(* IEC 61131-3 sources: AXOpen/src/components.festo.drives/ctrl/src/AxoCmmtAs (part 4) *)

            _AxisReference ?= AxisRef;

            IF(_AxisReference = NULL) THEN
                Messenger.Activate(     UINT#1690, eAxoMessageCategory#ProgrammingError);
                DriveStatus.Error.Id := UINT#1690;
                RETURN;
            END_IF;

            IF Enable THEN
                THIS.UpdateInputs(AxisRef);
                Valid := TRUE;
                Torque := THIS.ActualTorque;
            END_IF;
        END_METHOD

        ///<summary>
        /// This method returns in detail the status of the state diagram of the axis
        ///</summary>
        VAR INTERNAL
            MC_ReadStatusEnable_PV				: 	BOOL := FALSE;		//Enable - previous value
            MC_ReadStatusDone_PV				:	BOOL := FALSE;		//Done - previous value
            MC_ReadStatusStateNumber			: 	INT; 				//Call number of the method MC_ReadRealParameter
        END_VAR
        METHOD PUBLIC OVERRIDE MC_ReadStatus
            VAR_INPUT
                AxisRef             :   AXOpen.Components.Abstractions.Drives.IAxoAxisReference;
                Enable              :   BOOL;                       //  Get the value of the parameter continuously while enabled
            END_VAR
            VAR_OUTPUT
                Valid               :   BOOL;                       //  A valid output is available at the method
                Busy                :   BOOL;                       //  The method is not finished and new output values are to be expected
                Error               :   BOOL;                       //  Signals that an error has occurred within the method
                ErrorID             :   DINT;                       //  Error identification
                ErrorStop           :   BOOL;                       //  See state diagram
                Disabled            :   BOOL;                       //  See state diagram
                Stopping            :   BOOL;                       //  See state diagram
                Homing              :   BOOL;                       //  See state diagram
                Standstill          :   BOOL;                       //  See state diagram
                DiscreteMotion      :   BOOL;                       //  See state diagram
                ContinuousMotion    :   BOOL;                       //  See state diagram
                SynchronizedMotion  : BOOL;                       //  See state diagram
            END_VAR
            VAR
                _AxisReference :  REF_TO AXOpen.Components.Festo.Drives.AxoCmmtAsAxisReference;
                Dummy : BOOL;
            END_VAR

            _AxisReference ?= AxisRef;

            IF(_AxisReference = NULL) THEN
                Messenger.Activate(     UINT#1700, eAxoMessageCategory#ProgrammingError);
                DriveStatus.Error.Id := UINT#1700;
                RETURN;
            END_IF;

            IF Enable THEN
                THIS.UpdateInputs(AxisRef);
                Valid := TRUE;
                Error                   := _AxisReference^.Telegram111_In.ZSW1.faultPresent;
                ErrorID                 := _AxisReference^.Telegram111_In.Fault_Code;
                ErrorStop               := DriveState = AXOpen.Components.Drives.eAxoDriveState#ErrorStop;;
                Disabled                := DriveState = AXOpen.Components.Drives.eAxoDriveState#Disabled;
                Stopping                := DriveState = AXOpen.Components.Drives.eAxoDriveState#Stopping;
                Homing                  := DriveState = AXOpen.Components.Drives.eAxoDriveState#Homing;
                Standstill              := DriveState = AXOpen.Components.Drives.eAxoDriveState#Standstill;
                DiscreteMotion          := DriveState = AXOpen.Components.Drives.eAxoDriveState#DiscreteMotion;
                ContinuousMotion        := DriveState = AXOpen.Components.Drives.eAxoDriveState#ContinuousMotion;
                SynchronizedMotion      := DriveState = AXOpen.Components.Drives.eAxoDriveState#SynchronizedMotion;
            END_IF;
        END_METHOD

        ///<summary>
        /// This method returns in detail the status of the axis with respect to the motion currently in progress.
        ///</summary>
        VAR INTERNAL
            MC_ReadMotionStateEnable_PV     : 	BOOL := FALSE;		//Enable - previous value
            MC_ReadMotionStateErrorID       : 	WORD;
            MC_ReadMotionStateCycle			: 	ULINT;
            MC_ReadMotionStateValue			: 	LINT;
            MC_ReadMotionStateValid			: 	BOOL;
        END_VAR
        METHOD PUBLIC OVERRIDE MC_ReadMotionState
            VAR_INPUT
                AxisRef         :   AXOpen.Components.Abstractions.Drives.IAxoAxisReference;
                Enable          :   BOOL;                       //  Get the value of the parameter continuously while enabled
                Source          :   AXOpen.Components.Abstractions.Drives.eAxoSource;                 //  Defines the source of the relevant data: CommandedValue;SetValue, ActualValue.
            END_VAR
            VAR_OUTPUT
                Valid           :   BOOL;                       //  A valid output is available at the method
                Busy            :   BOOL;                       //  The method is not finished and new output values are to be expected
                Error           :   BOOL;                       //  Signals that an error has occurred within the method
                ErrorID         :   DINT;                       //  Error identification
                ConstantVelocity:   BOOL;                       //  Velocity is constant. Velocity may be 0. For the actual value a window is applicable (window is vendor specific)
                Accelerating    :   BOOL;                       //  Increasing the absolute value of the velocity
                Decelerating    :   BOOL;                       //  Decreasing the absolute value of the velocity
                DirectionPositive:  BOOL;                       //  Signals that the position is increasing
                DirectionNegative:  BOOL;                       //  Signals that the position is decreasing
            END_VAR
            VAR
                _AxisReference :  REF_TO AXOpen.Components.Festo.Drives.AxoCmmtAsAxisReference;
                Dummy : BOOL;
            END_VAR

            _AxisReference ?= AxisRef;

            IF(_AxisReference = NULL) THEN
                Messenger.Activate(     UINT#1710, eAxoMessageCategory#ProgrammingError);
                DriveStatus.Error.Id := UINT#1710;
                RETURN;
            END_IF;

            IF Enable THEN
                THIS.UpdateInputs(AxisRef);
                Valid := TRUE;
                Error                   := _AxisReference^.Telegram111_In.ZSW1.faultPresent;
                ErrorID                 := _AxisReference^.Telegram111_In.Fault_Code;
                ConstantVelocity        := FALSE;
                Accelerating            := _AxisReference^.Telegram111_In.ZSW1.axisAccelerates;
                Decelerating            := _AxisReference^.Telegram111_In.ZSW1.axisDecelerates;
                DirectionPositive       := _AxisReference^.Telegram111_In.POS_ZSW2.%X4;
                DirectionNegative       := _AxisReference^.Telegram111_In.POS_ZSW2.%X5;
             END_IF;
        END_METHOD

        ///<summary>
        /// This method reads information concerning an axis, like modes, inputs directly related to the axis,
        /// and certain status information.
        ///<summary>
        METHOD PUBLIC OVERRIDE MC_ReadAxisInfo
            VAR_INPUT
                AxisRef             :   AXOpen.Components.Abstractions.Drives.IAxoAxisReference;
                Enable              :   BOOL;                       //  Get the value of the parameter continuously while enabled
            END_VAR
            VAR_OUTPUT
                Valid               :   BOOL;                       //  A valid output is available at the method
                Busy                :   BOOL;                       //  The method is not finished and new output values are to be expected
                Error               :   BOOL;                       //  Signals that an error has occurred within the method
                ErrorID             :   DINT;                       //  Error identification
                HomeAbsSwitch       :   BOOL;                       //  Digital home switch input is active
                LimitSwitchPos      :   BOOL;                       //  Positive hardware end switch is active
                LimitSwitchNeg      :   BOOL;                       //  Negative hardware end switch is active
                Simulation          :   BOOL;                       //  Axis is in simulation mode (e.g. motor is simulated)
                CommunicationReady  :   BOOL;                         //  “Network” is initialized and ready for communication
                ReadyForPowerOn     :   BOOL;                       //  Drive is ready to be enabled (power on)
                PowerOn             :   BOOL;                       //  If TRUE shows that the power stage is switched ON
                IsHomed             :   BOOL;                       //  The absolute reference position is known for the axis (axis is homed)
                AxisWarning         :   BOOL;                       //  Warning(s) on the axis is present
            END_VAR
            VAR
                _AxisReference :  REF_TO AXOpen.Components.Festo.Drives.AxoCmmtAsAxisReference;
                Dummy : BOOL;
            END_VAR

            _AxisReference ?= AxisRef;

            IF(_AxisReference = NULL) THEN
                Messenger.Activate(     UINT#1720, eAxoMessageCategory#ProgrammingError);
                DriveStatus.Error.Id := UINT#1720;
                RETURN;
            END_IF;

            IF Enable THEN
                THIS.UpdateInputs(AxisRef);
                Valid := TRUE;
                Error                   := _AxisReference^.Telegram111_In.ZSW1.faultPresent;
                ErrorID                 := _AxisReference^.Telegram111_In.Fault_Code;
                HomeAbsSwitch           := FALSE;
                LimitSwitchPos          := _AxisReference^.Telegram111_In.POS_ZSW1.%X9;
                LimitSwitchNeg          := _AxisReference^.Telegram111_In.POS_ZSW1.%X8;
                Simulation              := FALSE;
                CommunicationReady      := FALSE;
                ReadyForPowerOn         := _AxisReference^.Telegram111_In.ZSW1.readyForSwitchOn;
                PowerOn                 := _AxisReference^.Telegram111_In.ZSW1.operationEnabled;
                IsHomed                 := _AxisReference^.Telegram111_In.ZSW1.homePosSet;
                AxisWarning             := _AxisReference^.Telegram111_In.ZSW1.warningActive;
            END_IF;
        END_METHOD

        ///<summary>
        /// This method presents general axis errors not relating to the methods.
        /// (for instance axis errors, drive errors, communication errors)
        ///</summary>
        VAR INTERNAL
            MC_ReadAxisErrorEnable_PV        : 	BOOL := FALSE;		//Enable - previous value
            MC_ReadAxisErrorErrorID          : 	DINT;
            MC_ReadAxisErrorCycle			: 	ULINT;
            MC_ReadAxisErrorValue			: 	LINT;
            MC_ReadAxisErrorValid			: 	BOOL;
            LastMessageCode :   ULINT;
        END_VAR
        METHOD PUBLIC OVERRIDE MC_ReadAxisError
            VAR_INPUT
                AxisRef         :   AXOpen.Components.Abstractions.Drives.IAxoAxisReference;
                Enable          :   BOOL;                       //  Get the value of the parameter continuously while enabled
            END_VAR
            VAR_OUTPUT
                Valid           :   BOOL;                       //  A valid output is available at the method
                Busy            :   BOOL;                       //  The method is not finished and new output values are to be expected
                Error           :   BOOL;                       //  Signals that an error has occurred within the method
                ErrorID         :   DINT;                       //  Error identification
                AxisErrorID     :   DWORD;                      //  The value of the axis error. These values are vendor specific
            END_VAR
            VAR
                _AxisReference :  REF_TO AXOpen.Components.Festo.Drives.AxoCmmtAsAxisReference;
                Dummy : BOOL;
                _category  :   AXOpen.Messaging.eAxoMessageCategory;
            END_VAR

            _AxisReference ?= AxisRef;

            IF(_AxisReference = NULL) THEN
                Messenger.Activate(     UINT#1730, eAxoMessageCategory#ProgrammingError);
                DriveStatus.Error.Id := UINT#1730;
                RETURN;
            END_IF;

            IF Enable AND NOT MC_ReadAxisErrorEnable_PV AND State = UINT#0 THEN
                _AxisReference^.Status.CurrentMotionTaskId := AXOpen.Components.Drives.eAxoMotionTaskId#Axo_ReadAxisError;
                _AxisReference^.Data.Cycle := _AxisReference^.Data.Cycle + ULINT#2;
                MC_ReadAxisErrorCycle := _AxisReference^.Data.Cycle ;
            END_IF;

            IF Enable THEN
                THIS.UpdateInputs(AxisRef);
                IF State = UINT#0 THEN
                    Busy := TRUE;
                    MC_ReadAxisErrorErrorID := DINT#0;
                    Parametrization.Inputs.Enable := FALSE;
                    State := UINT#310;
                END_IF;
                IF State = UINT#310 THEN
                    Busy := TRUE;
                    Parametrization.Inputs.Enable := TRUE;
                    Parametrization.Inputs.ReadWrite   := FALSE;
                    Parametrization.Inputs.ParameterNo := 12306;
                    Parametrization.Inputs.Subindex    := 0;
                    Parametrization.Inputs.AxisNo  := BYTE#1;
                    Parametrization.Inputs.HardwareId  := _AxisReference^.HWIDs.HW_ModuleAccessPoint;
                    IF Parametrization.Outputs.Done AND NOT Parametrization.Outputs.Error THEN
                        MC_ReadAxisErrorValid := TRUE;
                        MC_ReadAxisErrorValue := Parametrization.Outputs.ValueReadLINT;
                        State := UINT#311;
                    END_IF;
                    IF Parametrization.Outputs.Error THEN
                        Messenger.Activate(         UINT#1731, eAxoMessageCategory#Error);
                        MC_ReadAxisErrorErrorID :=  DINT#1731;
                        State := UINT#319;
                    END_IF;
                END_IF;
                IF State = UINT#311 THEN
                    Busy := TRUE;
                    Parametrization.Inputs.Enable := FALSE;
                    Parametrization.Inputs.ReadWrite   := FALSE;
                    IF  NOT Parametrization.Outputs.Done THEN
                        State := UINT#310;
                    END_IF;
                END_IF;
                IF State = UINT#319 THEN
                    Error := TRUE;
                END_IF;

                IF State>=UINT#310 AND State<UINT#317 THEN
                    IF _AxisReference^.Data.Cycle <> MC_ReadAxisErrorCycle THEN
                        _AxisReference^.Data.Cycle := _AxisReference^.Data.Cycle - ULINT#1;
                        State := UINT#319;
                    END_IF;
                END_IF;
                THIS.UpdateOutputs(AxisRef);
            END_IF;

            IF NOT Enable AND MC_ReadAxisErrorEnable_PV  THEN
                _AxisReference^.Status.CurrentMotionTaskId := AXOpen.Components.Drives.eAxoMotionTaskId#Axo_None;
                MC_ReadAxisErrorErrorID := DINT#0;
                MC_ReadAxisErrorCycle := ULINT#0;
                MC_ReadAxisErrorValid := FALSE;
                MC_ReadAxisErrorValue := LINT#0;
                State := UINT#0;
            END_IF;

            ErrorID := MC_ReadAxisErrorErrorID;
            Valid := MC_ReadAxisErrorValid;
            MC_ReadAxisErrorEnable_PV := Enable;

            Messenger.ActivateOnCondition(LastMessageCode,Enable AND Valid AND LastMessageCode = TO_ULINT(MC_ReadAxisErrorValue), eAxoMessageCategory#Error);
            // IF NOT Messenger.IsActive THEN
            IF Messenger.MessengerState = eAxoMessengerState#Idle THEN
                LastMessageCode := TO_ULINT(MC_ReadAxisErrorValue);
            END_IF;
        END_METHOD

        ///<summary>
        /// This method makes the transition from the state ‘ErrorStop’ to ‘Standstill’ or ‘Disabled’ by resetting all
        /// internal axis-related errors – it does not affect the output of the other methods.
        ///</summary>
        VAR INTERNAL
            MC_ResetExecute_PV					: 	BOOL := FALSE;		//Execute - previous value
            MC_ResetPower_PV					: 	BOOL := FALSE;		//Execute - previous value
        END_VAR
        METHOD PUBLIC OVERRIDE MC_Reset
            VAR_INPUT
                AxisRef         :   AXOpen.Components.Abstractions.Drives.IAxoAxisReference;
                Execute         :   BOOL;                       //  Resets all internal axis-related error
            END_VAR
            VAR_OUTPUT
                Done            :   BOOL;                       //  ‘Standstill’ or ‘Disabled’ state is reached
                Busy            :   BOOL;                       //  The method is not finished and new output values are to be expected
                Error           :   BOOL;                       //  Signals that an error has occurred within the method
                ErrorID         :   DINT;                       //  Error identification
            END_VAR
            VAR
                _AxisReference :  REF_TO AXOpen.Components.Festo.Drives.AxoCmmtAsAxisReference;
                Dummy : BOOL;
            END_VAR

            _AxisReference ?= AxisRef;

            IF(_AxisReference = NULL) THEN
                Messenger.Activate(     UINT#1740, eAxoMessageCategory#ProgrammingError);
                DriveStatus.Error.Id := UINT#1740;
                RETURN;
            END_IF;

            IF Execute AND NOT MC_ResetExecute_PV THEN
                _AxisReference^.Telegram111_Out.STW1.StartHoming := FALSE;
                _AxisReference^.Telegram111_Out.POS_STW1.MDI_MOD := FALSE;
                _AxisReference^.Telegram111_Out.POS_STW1.PosModulo := FALSE;
                _AxisReference^.Telegram111_Out.POS_STW1.NegModulo := FALSE;
                _AxisReference^.Telegram111_Out.POS_STW1.SetupMode := FALSE;
                _AxisReference^.Telegram111_Out.POS_STW1.MDI_Activate := FALSE;
                _AxisReference^.Telegram111_Out.POS_STW2.Trackingmode := FALSE;
                _AxisReference^.Telegram111_Out.POS_STW2.jog_inc := FALSE;
                _AxisReference^.Telegram111_Out.POS_STW1.travBlockBit0 := FALSE;
                _AxisReference^.Telegram111_Out.POS_STW1.travBlockBit1 := FALSE;
                _AxisReference^.Telegram111_Out.POS_STW1.travBlockBit2 := FALSE;
                _AxisReference^.Telegram111_Out.POS_STW1.travBlockBit3 := FALSE;
                _AxisReference^.Telegram111_Out.POS_STW1.travBlockBit4 := FALSE;
                _AxisReference^.Telegram111_Out.POS_STW1.travBlockBit5 := FALSE;
                _AxisReference^.Telegram111_Out.POS_STW1.travBlockBit6 := FALSE;
                _AxisReference^.Telegram111_Out.STW2.TravelToFixStop := FALSE;
                Parametrization.Inputs.Enable := FALSE;
                State := UINT#320;
            END_IF;

            IF Execute THEN
                THIS.UpdateInputs(AxisRef);

                IF State = UINT#320 THEN
                    Busy := TRUE;
                    THIS.Restore();
                    THIS.AxoReset_Task.Invoke(THIS);
                    State := UINT#321;
                END_IF;
                IF State = UINT#321 THEN
                    Busy := TRUE;
                    MC_ResetPower_PV := AxoPower_Task.IsSwitchedOn();
                    State := UINT#322;
                END_IF;
                IF State = UINT#322 THEN
                    Busy := TRUE;
                    THIS.AxoPower_Task.SwitchOff();
                    IF THIS.AxoPower_Task.IsSwitchedOff() THEN
                        State := UINT#323;
                    END_IF;
                END_IF;
                IF State = UINT#323 THEN
                    Busy := TRUE;
                    _AxisReference^.Telegram111_Out.STW1.acknowledgeFault := TRUE;
                    State := UINT#324;
                END_IF;
                IF State = UINT#324 THEN
                    Busy := TRUE;
                    IF  NOT _AxisReference^.Telegram111_In.ZSW1.faultPresent THEN
                        State := UINT#325;
                    END_IF;
                    IF  _AxisReference^.Telegram111_In.ZSW1.faultPresent  AND THIS.AxoReset_Task.Duration >=T#2S THEN
                        State := UINT#329;
                    END_IF;
                END_IF;
                IF State = UINT#325 THEN
                    Busy := TRUE;
                    IF MC_ResetPower_PV THEN
                        State := UINT#326;
                    ELSE
                        State := UINT#327;
                    END_IF;
                END_IF;
                IF State = UINT#326 THEN
                    Busy := TRUE;
                    THIS.AxoPower_Task.SwitchOn();
                    IF THIS.AxoPower_Task.IsSwitchedOn() THEN
                        State := UINT#327;
                    END_IF;
                END_IF;
                IF State = UINT#327 THEN
                    _AxisReference^.Telegram111_Out.STW1.acknowledgeFault := FALSE;
                    Done := TRUE;
                END_IF;
                IF State = UINT#329 THEN
                    _AxisReference^.Telegram111_Out.STW1.acknowledgeFault := FALSE;
                    Error := TRUE;
                    ErrorID := TO_DINT(_AxisReference^.Telegram111_In.Fault_Code);
                END_IF;
                THIS.UpdateOutputs(AxisRef);
            END_IF;

            IF NOT Execute AND MC_ResetExecute_PV THEN
                State := UINT#0;
            END_IF;

            MC_ResetExecute_PV := Execute;
        END_METHOD

        METHOD PUBLIC OVERRIDE Restore
            MC_PowerCycle                       := ULINT#0;
            MC_HomeExecute_PV					:= FALSE;
            MC_HomeErrorID					    := DINT#0;
            MC_HomeCycle					    := ULINT#0;
            MC_StopExecute_PV					:= FALSE;
            MC_StopErrorID					    := DINT#0;
            MC_StopCycle					    := ULINT#0;
            MC_HaltExecute_PV					:= FALSE;
            MC_HaltErrorID					    := DINT#0;
            MC_HaltCycle					    := ULINT#0;
            MC_MoveAbsoluteExecute_PV			:= FALSE;
            MC_MoveAbsoluteErrorID				:= DINT#0;
            MC_MoveAbsoluteCycle				:= ULINT#0;
            MC_MoveAbsoluteContinuousUpdate_SV  := FALSE;
            MC_MoveAbsolutePosition_PV          := LREAL#0.0;
            MC_MoveAbsoluteVelocity_PV          := LREAL#0.0;
            MC_MoveAbsoluteAcceleration_PV      := LREAL#0.0;
            MC_MoveAbsoluteDeceleration_PV      := LREAL#0.0;
            MC_MoveAbsoluteJerk_PV              := LREAL#0.0;
            MC_MoveAbsoluteDirection_PV         := AXOpen.Components.Abstractions.Drives.eAxoDriveDirection#CurrentDirection;
            MC_MoveRelativeExecute_PV			:= FALSE;
            MC_MoveRelativeErrorID				:= DINT#0;
            MC_MoveRelativeCycle				:= ULINT#0;
            MC_MoveRelativeContinuousUpdate_SV  := FALSE;
            MC_MoveRelativeDistance_PV          := LREAL#0.0;
            MC_MoveRelativeVelocity_PV          := LREAL#0.0;
            MC_MoveRelativeAcceleration_PV      := LREAL#0.0;
            MC_MoveRelativeDeceleration_PV      := LREAL#0.0;
            MC_MoveRelativeJerk_PV              := LREAL#0.0;
            MC_MoveAdditiveExecute_PV			:= FALSE;
            MC_MoveAdditiveErrorID				:= DINT#0;
            MC_MoveAdditiveCycle				:= ULINT#0;
            MC_MoveAdditiveContinuousUpdate_SV  := FALSE;
            MC_MoveAdditiveDistance_PV          := LREAL#0.0;
            MC_MoveAdditiveVelocity_PV          := LREAL#0.0;
            MC_MoveAdditiveAcceleration_PV      := LREAL#0.0;
            MC_MoveAdditiveDeceleration_PV      := LREAL#0.0;
            MC_MoveAdditiveJerk_PV              := LREAL#0.0;
            MC_MoveVelocityExecute_PV			:= FALSE;
            MC_MoveVelocityErrorID				:= DINT#0;
            MC_MoveVelocityCycle				:= ULINT#0;
            MC_MoveVelocityContinuousUpdate_SV  := FALSE;
            MC_MoveVelocityVelocity_PV          := LREAL#0.0;
            MC_MoveVelocityAcceleration_PV      := LREAL#0.0;
            MC_MoveVelocityDeceleration_PV      := LREAL#0.0;
            MC_MoveVelocityJerk_PV              := LREAL#0.0;
            MC_MoveVelocityDirection_PV         := AXOpen.Components.Abstractions.Drives.eAxoDriveDirection#CurrentDirection;
            MC_TorqueControlExecute_PV			:= FALSE;
            MC_TorqueControlErrorID				:= DINT#0;
            MC_TorqueControlCycle				:= ULINT#0;
            MC_TorqueControlContinuousUpdate_SV := FALSE;
            MC_TorqueControlTorque_PV           := LREAL#0.0;
            MC_TorqueControlTorqueRamp_PV       := LREAL#0.0;
            MC_TorqueControlPositionLimit_PV    := LREAL#0.0;
            MC_TorqueControlVelocity_PV         := LREAL#0.0;
            MC_TorqueControlAcceleration_PV     := LREAL#0.0;
            MC_TorqueControlDeceleration_PV     := LREAL#0.0;
            MC_TorqueControlJerk_PV             := LREAL#0.0;
            MC_TorqueControlDirection_PV        := AXOpen.Components.Abstractions.Drives.eAxoDriveDirection#CurrentDirection;
            MC_SetPositionExecute_PV			:= FALSE;
            MC_SetPositionErrorID				:= DINT#0;
            MC_SetPositionCycle					:= ULINT#0;
            MC_SetPositionActualPosition        := LINT#0;
            MC_ReadParameterEnable_PV           := FALSE;
            MC_ReadParameterErrorID             := DINT#0;
            MC_ReadParameterCycle			    := ULINT#0;
            MC_ReadParameterValue			    := LINT#0;
            MC_ReadParameterValid			    := FALSE;
            MC_ReadRealParameterEnable_PV       := FALSE;
            MC_ReadRealParameterErrorID         := DINT#0;
            MC_ReadRealParameterCycle			:= ULINT#0;
            MC_ReadRealParameterValue			:= REAL#0.0;
            MC_ReadRealParameterValid			:= FALSE;
            MC_ReadBoolParameterEnable_PV       := FALSE;
            MC_ReadBoolParameterErrorID         := DINT#0;
            MC_ReadBoolParameterCycle			:= ULINT#0;
            MC_ReadBoolParameterValue			:= FALSE;
            MC_ReadBoolParameterValid			:= FALSE;
            MC_WriteParameterExecute_PV         := FALSE;
            MC_WriteParameterErrorID            := DINT#0;
            MC_WriteParameterCycle			    := ULINT#0;
            MC_WriteRealParameterExecute_PV     := FALSE;
            MC_WriteRealParameterErrorID        := DINT#0;
            MC_WriteRealParameterCycle			:= ULINT#0;
            MC_WriteBoolParameterExecute_PV     := FALSE;
            MC_WriteBoolParameterErrorID        := DINT#0;
            MC_WriteBoolParameterCycle			:= ULINT#0;
            MC_ReadDigitalInputEnable_PV        := FALSE;
            MC_ReadDigitalInputErrorID          := DINT#0;
            MC_ReadDigitalInputCycle			:= ULINT#0;
            MC_ReadDigitalInputValue			:= FALSE;
            MC_ReadDigitalInputValid			:= FALSE;
            MC_ReadDigitalOutputEnable_PV       := FALSE;
            MC_ReadDigitalOutputErrorID         := DINT#0;
            MC_ReadDigitalOutputCycle			:= ULINT#0;
            MC_ReadDigitalOutputValue			:= FALSE;
            MC_ReadDigitalOutputValid			:= FALSE;
            MC_WriteDigitalOutputExecute_PV     := FALSE;
            MC_WriteDigitalOutputErrorID        := DINT#0;
            MC_WriteDigitalOutputCycle			:= ULINT#0;
            MC_ReadStatusEnable_PV				:= FALSE;
            MC_ReadStatusDone_PV				:= FALSE;
            MC_ReadStatusStateNumber			:= INT#0;
            MC_ReadMotionStateEnable_PV         := FALSE;
            MC_ReadMotionStateErrorID           := WORD#0;
            MC_ReadMotionStateCycle			    := ULINT#0;
            MC_ReadMotionStateValue			    := LINT#0;
            MC_ReadMotionStateValid			    := FALSE;
            MC_ReadAxisErrorEnable_PV           := FALSE;
            MC_ReadAxisErrorErrorID             := DINT#0;
            MC_ReadAxisErrorCycle			    := ULINT#0;
            MC_ReadAxisErrorValue			    := LINT#0;
            MC_ReadAxisErrorValid			    := FALSE;
            LastMessageCode                     := ULINT#0;
            MC_ResetExecute_PV				    := FALSE;
            MC_ResetPower_PV				    := FALSE;

            AxisRefExt.Data.Cycle              := ULINT#0;
            State                               := UINT#0;
            DriveStatus.Action.Id := UINT#0;
            DriveStatus.Error.Id  := UINT#0;
            Messenger.Restore();
            TaskMessenger.Restore();

            //AxoPower_Task.Restore();
            AxoStop_Task.Restore();
            AxoHalt_Task.Restore();
            AxoHome_Task.Restore();
            AxoMoveAbsolute_Task.Restore();
            AxoMoveRelative_Task.Restore();
            AxoMoveAdditive_Task.Restore();
            AxoMoveVelocity_Task.Restore();
            AxoTorqueControl_Task.Restore();
            AxoSetPosition_Task.Restore();
            AxoSetOverride_Task.SwitchOff();
            AxoReadParameter_Task.SwitchOff();
            AxoReadRealParameter_Task.SwitchOff();
            AxoReadBoolParameter_Task.SwitchOff();
            AxoWriteParameter_Task.Restore();
            AxoWriteRealParameter_Task.Restore();
            AxoWriteBoolParameter_Task.Restore();
            AxoReadDigitalInput_Task.SwitchOff();
            AxoReadDigitalOutput_Task.SwitchOff();
            AxoWriteDigitalOutput_Task.Restore();
            AxoReadActualPosition_Task.SwitchOff();
            AxoReadActualVelocity_Task.SwitchOff();
            AxoReadActualTorque_Task.SwitchOff();
            AxoReadStatus_Task.SwitchOff();
            AxoReadMotionState_Task.SwitchOff();
            AxoReadAxisInfo_Task.SwitchOff();
            AxoReadAxisError_Task.SwitchOff();
            AxoReset_Task.Restore();
            AxoJogPositive.RemoteSwitchOn := FALSE;
            AxoJogPositive.StartMotion := FALSE;
            AxoJogPositive.StopMotion := FALSE;
            AxoJogNegative.RemoteSwitchOn := FALSE;
            AxoJogNegative.StartMotion := FALSE;
            AxoJogNegative.StopMotion := FALSE;
            Parametrization.Restore();

            AxisRefExt.Telegram111_Out.STW1.activateTraversing := FALSE;
            AxisRefExt.Telegram111_Out.STW1.StartHoming := FALSE;
            AxisRefExt.Telegram111_Out.POS_STW1.MDI_MOD := FALSE;
            AxisRefExt.Telegram111_Out.POS_STW1.PosModulo := FALSE;
            AxisRefExt.Telegram111_Out.POS_STW1.NegModulo := FALSE;
            AxisRefExt.Telegram111_Out.POS_STW1.SetupMode := FALSE;
            AxisRefExt.Telegram111_Out.POS_STW1.MDI_Activate := FALSE;
            AxisRefExt.Telegram111_Out.POS_STW2.Trackingmode := FALSE;
            AxisRefExt.Telegram111_Out.POS_STW2.jog_inc := FALSE;
            AxisRefExt.Telegram111_Out.POS_STW1.travBlockBit0 := FALSE;
            AxisRefExt.Telegram111_Out.POS_STW1.travBlockBit1 := FALSE;
            AxisRefExt.Telegram111_Out.POS_STW1.travBlockBit2 := FALSE;
            AxisRefExt.Telegram111_Out.POS_STW1.travBlockBit3 := FALSE;
            AxisRefExt.Telegram111_Out.POS_STW1.travBlockBit4 := FALSE;
            AxisRefExt.Telegram111_Out.POS_STW1.travBlockBit5 := FALSE;
            AxisRefExt.Telegram111_Out.POS_STW1.travBlockBit6 := FALSE;
            AxisRefExt.Telegram111_Out.STW2.TravelToFixStop := FALSE;

            SUPER.Restore();

            RestoreTask.DoneWhen(TRUE);
        END_METHOD
    END_CLASS
END_NAMESPACE

(* ---- AxoCmmtAsAxisData.st ---- *)
NAMESPACE AXOpen.Components.Festo.Drives
    {S7.extern=ReadWrite}
    CLASS AxoCmmtAsAxisData
        VAR PUBLIC
            hwID                        :   WORD;
            hwIdModuleAccessPoint       :   WORD;
            hwIdTelegram111             :   WORD;
            hwIdTelegram750             :   WORD;
            Cycle                       :   ULINT;
            OverrideVelocityFactor		:	LREAL := 1.0;	//LREAL value to be written
            OverrideAccelerationFactor	:	LREAL := 1.0;	//LREAL value to be written
            OverrideJerkFactor			:	LREAL := 1.0;	//LREAL value to be written
        END_VAR
    END_CLASS
END_NAMESPACE

(* ---- AxoCmmtAsAxisReference.st ---- *)
// USING AXOpen.Components.Drives;

NAMESPACE AXOpen.Components.Festo.Drives
    {S7.extern=ReadWrite}
    CLASS AxoCmmtAsAxisReference IMPLEMENTS AXOpen.Components.Abstractions.Drives.IAxoAxisReference
        VAR PUBLIC
            Telegram111_In  :   AXOpen.Components.Festo.Drives.PROFIdriveTelegram_111_IN;
            Telegram111_Out :   AXOpen.Components.Festo.Drives.PROFIdriveTelegram_111_OUT;
            Telegram750_In  :   AXOpen.Components.Festo.Drives.PROFIdriveTelegram_750_IN;
            Telegram750_Out :   AXOpen.Components.Festo.Drives.PROFIdriveTelegram_750_OUT;
            Data            :   AXOpen.Components.Festo.Drives.AxoCmmtAsAxisData;
            Config          :   AXOpen.Components.Drives.AxoDrive_Config;
            Status          :   AXOpen.Components.Drives.AxoDrive_Status;
        END_VAR
    END_CLASS
END_NAMESPACE

(* ---- AxoCmmtAsFieldBusIn.st ---- *)
NAMESPACE AXOpen.Components.Festo.Drives
    {S7.extern=ReadWrite}
    CLASS AxoCmmtAsFieldBusIn
        (******************* Drive configuration  ***********************
        Master communication; Fieldbus settings:

                Profile type: * free configurable mode*
                    Configuration of realtime channel:
                        realtime input (configured feedback values):	    (9words)
                                P-0-4078 Fieldbus status WORD               (2bytes)
                                S-0-0051 Position feedback 1 value          (4bytes)
                                S-0-0040 Veloccity feedback value           (4bytes)
                                S-0-0390 Diagnostig message number          (4bytes)
                                S-0-0144 Signal status  word			    (2bytes)
                                S-0-0084 Actual torque/force value          (2bytes)
                        realtime output (configured command values):		(13words)
                                P-0-4077 Fieldbus control WORD              (2bytes)
                                S-0-0282 Positioning command value          (4bytes)
                                S-0-0259 Positioning velocity value         (4bytes)
                                S-0-0260 Positioning Accelelration          (4bytes)
                                S-0-0359 Positioning Deceleration           (4bytes)
                                S-0-0145 Signal control word                (2bytes)
                                S-0-0080 Torque/force command value		    (2bytes)
                                S-0-0193 Positioning jerk                   (4bytes)
                General settings:
                        S-0-0027, Configuration list signal control word -> Number 0; Content S-0-0393
                        S-0-0329, Assign list signal control word -> Number 0; Content 2
                        Primary operation mode: Drive controlled positioning, encoder 1 (without axis control word)
                        Secondary operation mode: Torque/force control
        *)
        VAR PUBLIC
            PhaseAcknowledgeBit0		:	BOOL;		//Operating mode acknowledge bit 0
            PhaseAcknowledgeBit1 		:	BOOL;		//Operating mode acknowledge bit 1
            InReference 				:	BOOL;		//In reference
            InStandstill 				:	BOOL;		//In standstill
            SetpointReached				:	BOOL;		//Setpoint reached
            CommandChangeBit 			:	BOOL;		//Command change bit
            OperatingModeError 			:	BOOL;		//Operating mode_error
            StatusSetpointProcess 		:	BOOL;		//Status setpoint processing
            ActualOperatingModeBit0 	:	BOOL;		//Actual_operating mode bit 0
            ActualOperatingModeBit1 	:	BOOL;		//Actual_operating mode bit 1
            SetpointAcknowledge 		:	BOOL;		//Setpoint acknowledge
            MessageZKL3 				:	BOOL;		//Message ZKL3
            WarningZKL2 				:	BOOL;		//Warning ZKL2
            DriveErrorZKL1 				:	BOOL;		//Drive Error ZKL1
            ReadyToOperateBit0 			:	BOOL;		//Ready to operate bit 0
            ReadyToOperateBit1 			:	BOOL;		//Ready to operate bit 1
            S_0_0051_ActualPosition		:	DWORD;		//Actual position
            S_0_0040_ActualVelocity		:	DWORD;		//Actual velocity
            S_0_0390_Diagnosis			:	DWORD;		//Diagnosis
            S_0_0144_SignalStatusWord	:	WORD;		//Signal status word
            S_0_0084_ActualTorque 		:	WORD;		//Actual torque
        END_VAR
    END_CLASS

END_NAMESPACE

(* ---- AxoCmmtAsFieldBusOut.st ---- *)
NAMESPACE AXOpen.Components.Festo.Drives
    {S7.extern=ReadWrite}
    CLASS AxoCmmtAsFieldBusOut
        (******************* Drive configuration  ***********************
        Master communication; Fieldbus settings:

                Profile type: * free configurable mode*
                    Configuration of realtime channel:
                        realtime input (configured feedback values):	    (9words)
                                P-0-4078 Fieldbus status WORD               (2bytes)
                                S-0-0051 Position feedback 1 value          (4bytes)
                                S-0-0040 Veloccity feedback value           (4bytes)
                                S-0-0390 Diagnostig message number          (4bytes)
                                S-0-0144 Signal status  word			    (2bytes)
                                S-0-0084 Actual torque/force value          (2bytes)
                        realtime output (configured command values):		(13words)
                                P-0-4077 Fieldbus control WORD              (2bytes)
                                S-0-0282 Positioning command value          (4bytes)
                                S-0-0259 Positioning velocity value         (4bytes)
                                S-0-0260 Positioning Accelelration          (4bytes)
                                S-0-0359 Positioning Deceleration           (4bytes)
                                S-0-0145 Signal control word                (2bytes)
                                S-0-0080 Torque/force command value		    (2bytes)
                                S-0-0193 Positioning jerk                   (4bytes)
                General settings:
                        S-0-0027, Configuration list signal control word -> Number 0; Content S-0-0393
                        S-0-0329, Assign list signal control word -> Number 0; Content 2
                        Primary operation mode: Drive controlled positioning, encoder 1 (without axis control word)
                        Secondary operation mode: Torque/force control
        *)
        VAR PUBLIC
            SetpointAcceptance 				:	BOOL;			//Setpoint acceptance
            OperatingModeSet 				:	BOOL;			//Operating mode set
            DriveToZeroPoint 				:	BOOL;			//Drive to zero point
            AbsoluteRelative 				:	BOOL;			//Position absolute = 0 or relative = 1
            ImmediateBlockChange 			:	BOOL;			//Immediate change
            ErrorDelete 					:	BOOL;			//Clear error
            JogForward 						:	BOOL;			//Jog forward
            JogBackward 					:	BOOL;			//Jog backward
            SetOperatingModeBit0 			:	BOOL;			//Setpoint operating mode_bit0
            SetOperatingModeBit1 			:	BOOL;			//Setpoint operating mode_bit1
            Iposync 						:	BOOL;			//Only in cycl. pos. control
            DriveHalt 						:	BOOL;			//Drive halt
            DriveEnable 					:	BOOL;			//Drive enable
            DriveOn 						:	BOOL;			//Drive on
            S_0_0282_CommandPosition		: 	DWORD;			//Command position
            S_0_0259_CommandVelocity		: 	DWORD;          //Command velocity
            S_0_0260_CommandAcceleration	: 	DWORD;          //Command acceleration
            S_0_0359_CommandDecceleration	: 	DWORD;          //Command decceleration
            S_0_0145_SignalControlWord		: 	WORD;           //Signal control word
            S_0_0080_TorqueForceCommand     :   WORD;           //Torque/force command value
            S_0_0193_CommandJerk            :   DWORD;          //Command jerk
        END_VAR
    END_CLASS
END_NAMESPACE
